SUBAPPLICATION OPC_SUB_1 (* Subapplication Type *)
  (* Standard: 61499-2 *)
  (* Version 1.0, 2022-03-09, Maximilian Scharf *)
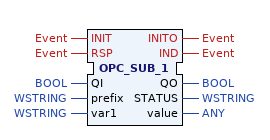
  EVENT_INPUT
    INIT;
    RSP;
  END_EVENT
  EVENT_OUTPUT
    INITO;
    IND;
  END_EVENT
  VAR_INPUT
    QI : BOOL;
    prefix : WSTRING;
    var1 : WSTRING;
  END_VAR
  VAR_OUTPUT
    QO : BOOL;
    STATUS : WSTRING;
    value : ANY;
  END_VAR
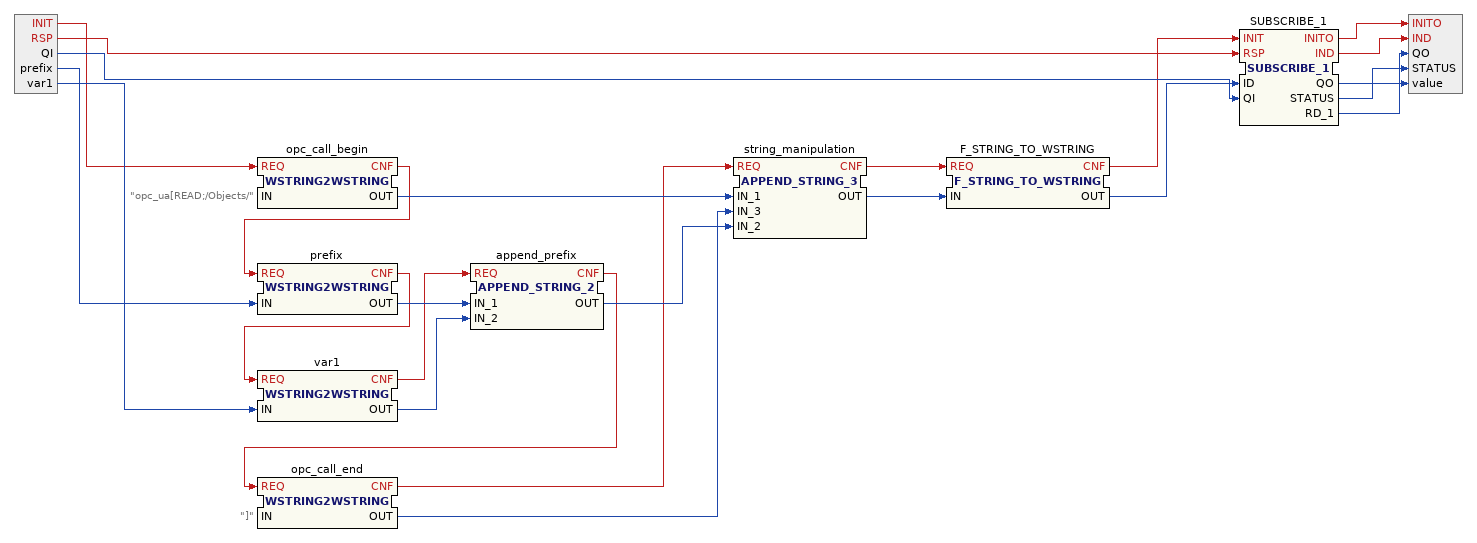
  FBS
    opc_call_begin : WSTRING2WSTRING(IN := "opc_ua[READ;/Objects/");
    F_STRING_TO_WSTRING : F_STRING_TO_WSTRING;
    string_manipulation : APPEND_STRING_3;
    opc_call_end : WSTRING2WSTRING(IN := "]");
    var1 : WSTRING2WSTRING;
    SUBSCRIBE_1 : SUBSCRIBE_1;
    append_prefix : APPEND_STRING_2;
    prefix : WSTRING2WSTRING;
  END_FBS
  EVENT_CONNECTIONS
    string_manipulation.CNF TO F_STRING_TO_WSTRING.REQ;
    opc_call_end.CNF TO string_manipulation.REQ;
    INIT TO opc_call_begin.REQ;
    F_STRING_TO_WSTRING.CNF TO SUBSCRIBE_1.INIT;
    SUBSCRIBE_1.INITO TO INITO;
    RSP TO SUBSCRIBE_1.RSP;
    SUBSCRIBE_1.IND TO IND;
    opc_call_begin.CNF TO prefix.REQ;
    prefix.CNF TO var1.REQ;
    var1.CNF TO append_prefix.REQ;
    append_prefix.CNF TO opc_call_end.REQ;
  END_CONNECTIONS
  DATA_CONNECTIONS
    opc_call_begin.OUT TO string_manipulation.IN_1;
    string_manipulation.OUT TO F_STRING_TO_WSTRING.IN;
    opc_call_end.OUT TO string_manipulation.IN_3;
    var1 TO var1.IN;
    F_STRING_TO_WSTRING.OUT TO SUBSCRIBE_1.ID;
    SUBSCRIBE_1.QO TO QO;
    SUBSCRIBE_1.STATUS TO STATUS;
    SUBSCRIBE_1.RD_1 TO value;
    QI TO SUBSCRIBE_1.QI;
    prefix TO prefix.IN;
    prefix.OUT TO append_prefix.IN_1;
    var1.OUT TO append_prefix.IN_2;
    append_prefix.OUT TO string_manipulation.IN_2;
  END_CONNECTIONS
END_SUBAPPLICATION
